TYPE "UDT_ZC_RECETA_CIP_SOSA_ENJ"
VERSION : 0.1
   STRUCT
      TiempoEmpujeADestino : Int;   // SOSA ENJ. Tiempo de empuje a destino
      TiempoMaxVaciadoDestino : Int;   // SOSA ENJ. Tiempo Max vaciado destino
      TiempoEmpujeDestinoACIP : Int;   // SOSA ENJ. Tiempoi empuje desde equipo a CIP
      TiempoMaxEnjuague : Int;   // SOSA ENJ. Tiempo Maximo Enjuague
      TiempoEnjuagueConConductividad : Int;   // SOSA ENJ. Tiempo enjuague con conductividad
      ReservaInt_1 : Int;   // SOSA ENJ.
      ReservaInt_2 : Int;   // SOSA ENJ.
      TemperaturaEnjuague : Real;   // SOSA ENJ. Temperatura Enjuague
      TemperaturaHisteresis : Real;   // SOSA ENJ. Temperatura Enjuague Histeresis
      ConductividadDrenaje : Real;   // SOSA ENJ. Conductividad para Drenaje
      ConductividadEnjuagueOk : Real;   // SOSA ENJ. Conductividad para Enjuague OK
      ConductividadDrenajeAguaRecup : Real;   // SOSA ENJ. Conductividad para drenaje/agua recup.
      ProcentajeEnvioDQO : Real;   // SOSA ENJ. Porcentaje de tiempo de envio a DQO
   END_STRUCT;

END_TYPE

